(* CODESYS project DosingMachine (4).project

Project tree, tasks and I/O mapping:
  Device : CODESYS Control Win V3 x64, 3S - Smart Software Solutions GmbH, version 3.5.12.20
    application Application
      libraries: Standard, * (System); Util, * (System)
      task MainTask (cyclic, interval t#20ms, priority 1) calls DosingMain
      task VISU_TASK (cyclic, interval 100 ms, priority 31) calls VisuElems.Visu_Prg
      function block Timer [LD]
      function block DosingBlock [ST]
      program DosingMain [CFC]: Animatoin
      function block FSM [ST]
      visualisation Visualization
      image pool ImagePool
  text list GlobalTextList
  5ce3da45-db07-42e7-a21c-a00fff4ed8f6|E:\MyFiles\VideoShooting\CircuitBreakers\Slides\11.A to Z Project #2\PLC Porgramming\Motor 5.png
  5ce3da45-db07-42e7-a21c-a00fff4ed8f6|E:\MyFiles\VideoShooting\CircuitBreakers\Slides\11.A to Z Project #2\PLC Porgramming\helezon.png
  5ce3da45-db07-42e7-a21c-a00fff4ed8f6|E:\MyFiles\VideoShooting\CircuitBreakers\Slides\11.A to Z Project #2\helezon.png
  5ce3da45-db07-42e7-a21c-a00fff4ed8f6|E:\MyFiles\VideoShooting\CircuitBreakers\Slides\11.A to Z Project #2\PLC Porgramming\ELAVATOR 9 METRE - Kopya.PNG
  5ce3da45-db07-42e7-a21c-a00fff4ed8f6|E:\MyFiles\VideoShooting\CircuitBreakers\Slides\11.A to Z Project #2\Motor 5green.png
  5ce3da45-db07-42e7-a21c-a00fff4ed8f6|E:\MyFiles\VideoShooting\CircuitBreakers\Slides\11.A to Z Project #2\PLC Porgramming\Motor 5green.png
  5ce3da45-db07-42e7-a21c-a00fff4ed8f6|E:\MyFiles\VideoShooting\CircuitBreakers\Slides\11.A to Z Project #2\PLC Porgramming\Motor 5red.png
  5ce3da45-db07-42e7-a21c-a00fff4ed8f6|E:\MyFiles\VideoShooting\CircuitBreakers\Slides\11.A to Z Project #2\PLC Porgramming\ELAVATOR 9 METREFlip.png
  5ce3da45-db07-42e7-a21c-a00fff4ed8f6|E:\MyFiles\VideoShooting\CircuitBreakers\Slides\11.A to Z Project #2\PLC Porgramming\helezonFlip.png
  5ce3da45-db07-42e7-a21c-a00fff4ed8f6|E:\MyFiles\VideoShooting\CircuitBreakers\Slides\11.A to Z Project #2\PLC Porgramming\Silo.png
  5ce3da45-db07-42e7-a21c-a00fff4ed8f6|E:\MyFiles\VideoShooting\CircuitBreakers\Slides\11.A to Z Project #2\PLC Porgramming\Motor 5Flip.png
  5ce3da45-db07-42e7-a21c-a00fff4ed8f6|E:\MyFiles\VideoShooting\CircuitBreakers\Slides\11.A to Z Project #2\PLC Porgramming\Motor 5greenFlip.png
  5ce3da45-db07-42e7-a21c-a00fff4ed8f6|E:\MyFiles\VideoShooting\CircuitBreakers\Slides\11.A to Z Project #2\PLC Porgramming\Motor 5redflip.png
*)

// Device/Application/DosingMain
PROGRAM DosingMain
VAR
	Elev1Coil		:BOOL;
	Elev2Coil		:BOOL;
	Spiral1Coil		:BOOL;
	Spiral2Coil		:BOOL;
	MixerCoil		:BOOL;
	MixerGateCoil	:BOOL;
	
	Elev1OVLD		:BOOL;
	Elev2OVLD		:BOOL;
	SPiral1OVLD		:BOOL;
	Spiral2OVLD		:BOOL;
	MixerOVLD		:BOOL;
	EMGC			:BOOL;
	X: BOOL;
	StartDosing		:BOOL;
	StopDosing		:BOOL;
	FillSilo1		:BOOL;
	FillSilo2		:BOOL;
	
	Spiral1Freq		:INT;
	Spiral2Freq		:INT;
	MixerFreq		:INT;
	
	
	Silo1Weight		:INT;
	Silo2Weight		:INT;
	
	Silo1Required	:INT;
	Silo2Required	:INT;
	

	Silo1Dosing: DosingBlock;
	Silo2Dosing: DosingBlock;
	TheMaestro: FSM;
	Timing: Timer;
	LIN_TRAFO_0: lin_trafo;
	Silo1: LIN_TRAFO;
	Silo1Animation: WORD;
	Silo1AnimationScale: WORD;
	Silo2: LIN_TRAFO;
	Silo2Animation: WORD;
	Silo2AnimationScale: WORD;
END_VAR
VAR // added by the converter: edge detectors and wires of the graphical bodies
    _w1, _w2, _w3, _w16 : BOOL;
    _w4, _w5, _w6, _w7, _w8, _w9, _w10, _w11, _w12, _w13, _w14, _w15 : ANY;
END_VAR

Spiral2Coil := Silo2Dosing.MotorCoil;
MixerGateCoil := _w1;
_w3 := _w2 OR MixerOVLD;
Elev1Coil := FillSilo1;
Elev2Coil := FillSilo2;
Animatoin();
Silo1Dosing(
    StartDosing := _w4,
    StopDosing := StopDosing,
    Weight := Silo1Weight,
    RequiredProduct := Silo1Required); // DosingBlock
Spiral1Coil := Silo1Dosing.MotorCoil;
(* _w3 OR EMGC; result not used *)
Timing(MixerTimerActivate := _w5, GateTimerActivate := _w6, MixerPreSet := t#20s, GatePreSet := T#20s); // Timer
TheMaestro(
    Start := StartDosing,
    Stop := StopDosing,
    EMGC := _w7,
    Silo1DoseDone := _w8,
    Silo2DoseDone := _w9,
    Silo1NotEnough := _w10,
    Silo2NotEnough := _w11,
    FillBusy := _w12,
    MixerTimerDone := _w13,
    GateTimerDone := _w14); // FSM
Silo2Dosing(
    StartDosing := _w15,
    StopDosing := StopDosing,
    Weight := Silo2Weight,
    RequiredProduct := Silo2Required); // DosingBlock
_w12 := FillSilo1 OR FillSilo2;
MixerCoil := _w16;
_w2 := SPiral1OVLD OR Spiral2OVLD;

ACTION Animatoin:
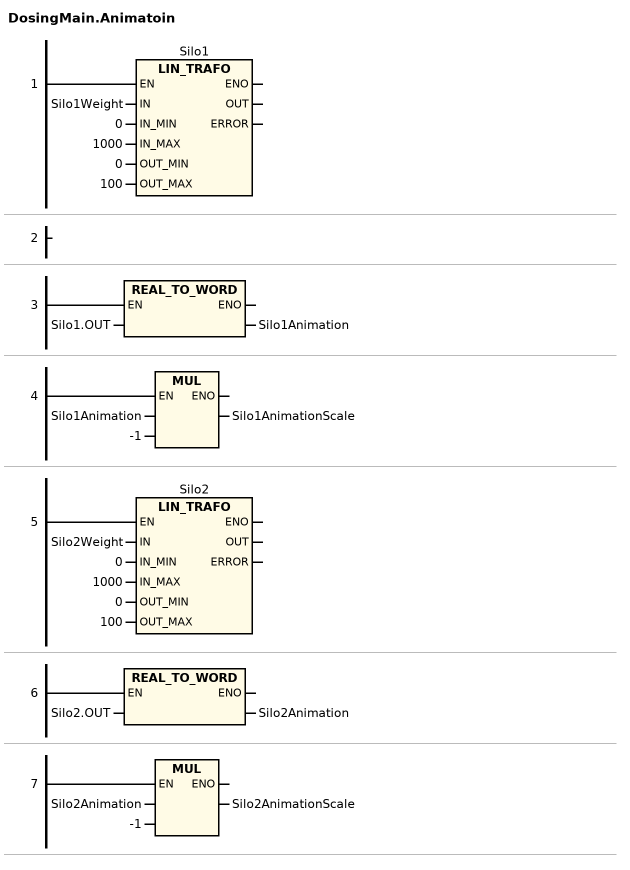
// NETWORK 1
Silo1(IN := Silo1Weight, IN_MIN := 0, IN_MAX := 1000, OUT_MIN := 0, OUT_MAX := 100); // LIN_TRAFO

// NETWORK 2

// NETWORK 3
Silo1Animation := REAL_TO_WORD(Silo1.OUT);

// NETWORK 4
Silo1AnimationScale := Silo1Animation * -1;

// NETWORK 5
Silo2(IN := Silo2Weight, IN_MIN := 0, IN_MAX := 1000, OUT_MIN := 0, OUT_MAX := 100); // LIN_TRAFO

// NETWORK 6
Silo2Animation := REAL_TO_WORD(Silo2.OUT);

// NETWORK 7
Silo2AnimationScale := Silo2Animation * -1;
END_ACTION

END_PROGRAM

// Device/Application/DosingBlock
FUNCTION_BLOCK DosingBlock
VAR_INPUT
	StartDosing : BOOL;
	StopDosing	: BOOL;
	Weight		:INT;
	RequiredProduct : INT;
	
END_VAR
VAR_OUTPUT
	MotorCoil        :BOOL;
	Extracted		 :INT;
	Busy			 :BOOL;
	Done			 :BOOL;
	NotEnough		 :BOOL;
END_VAR
VAR
	WeightSaved  : INT;
	StartTrig: R_TRIG;
END_VAR

StartTrig(CLK:=StartDosing , Q=> );

IF StartTrig.Q = 1 AND NotEnough=0 AND StopDosing=0 THEN
	WeightSaved := Weight ;
	MotorCoil:=1;
	Busy  :=1;
	Done :=0;
	
END_IF

IF Busy=1 THEN

Extracted :=	WeightSaved-Weight ;
IF Extracted>=RequiredProduct THEN
	MotorCoil :=0;
	Busy:=0;
	Done:=1;
END_IF
END_IF




IF RequiredProduct > Weight AND BUSY=0 THEN
	NotEnough:=1;
ELSE
	NotEnough:=0;
	
END_IF

IF StopDosing =1 THEN
	MotorCoil:=0;
	Busy:=0;
	Done:=1;
	
END_IF

END_FUNCTION_BLOCK

// Device/Application/Timer
FUNCTION_BLOCK Timer
VAR_INPUT
	MixerTimerActivate : BOOL;
	GateTimerActivate  :BOOL;
	MixerPreSet			:TIME;
	GatePreSet 			:TIME;
END_VAR
VAR_OUTPUT
	MixerTimerDone : BOOL;
	GateTimerDone   :BOOL;
END_VAR
VAR
	MixerTimer: TON;
	GateTimer: TON;
END_VAR

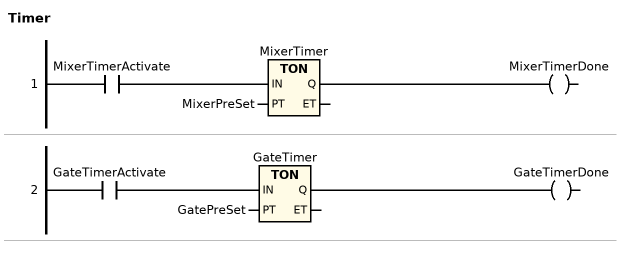
// NETWORK 1
MixerTimer(IN := MixerTimerActivate, PT := MixerPreSet); // TON
MixerTimerDone := MixerTimer.Q;

// NETWORK 2
GateTimer(IN := GateTimerActivate, PT := GatePreSet); // TON
GateTimerDone := GateTimer.Q;

END_FUNCTION_BLOCK

// Device/Application/FSM
FUNCTION_BLOCK FSM
VAR_INPUT
	Start 			:BOOL;
	Stop  			:BOOL;
	EMGC  			:BOOL;
	Silo1DoseDone 	:BOOL;
	Silo2DoseDone   :BOOL;
	Silo1NotEnough  :BOOL;
	Silo2NotEnough  :BOOL;
	FillBusy		:BOOL;
	MixerTimerDone  :BOOL;
	GateTimerDone	:BOOL;
	
END_VAR
VAR_OUTPUT
	Dose1BlockActivate  : BOOL;
	Dose2BlockActivate  :BOOL;
	MixerCoil		    :BOOL;
	GateCoil			:BOOL;
	MixerTimerActivate  :BOOL;
	GateTimerActivate   :BOOL;
	NotReady 			:BOOL;
	Stage				:INT;
END_VAR
VAR
	StartTrigger: R_TRIG;
	WeightSaved : INT;
	Silo1DoneTirg: R_TRIG;
	Silo2DoneTrig: R_TRIG;
END_VAR

StartTrigger(CLK:= Start , Q=> );
 
Silo1DoneTirg(CLK:= Silo1DoseDone  , Q=> );

 Silo2DoneTrig(CLK:= Silo2DoseDone , Q=> );
CASE Stage OF
	
0:
IF StartTrigger.Q = 1 AND NotReady=0 THEN
	Stage:=1;
END_IF

1:
Dose1BlockActivate:=1;
IF Silo1DoneTirg.Q =1 THEN
	Dose1BlockActivate:=0;
	Stage:=2;
END_IF

2:

Dose2BlockActivate:=1;
IF Silo2DoneTrig.Q =1 THEN
	Dose2BlockActivate:=0;
	Stage:=3;
END_IF


3:

MixerCoil:=1;
MixerTimerActivate:=1;

IF MixerTimerDone =1 THEN
MixerCoil:=0;
MixerTimerActivate:=0;	
Stage :=4;
END_IF

4:

GateCoil :=1 ;
GateTimerActivate := 1;
IF GateTimerDone =1 THEN
GateCoil :=0 ;	
GateTimerActivate := 0;
Stage:=0;

END_IF
END_CASE


IF EMGC OR Silo1NotEnough OR Silo2NotEnough OR FillBusy  OR STOP THEN
	NotReady :=1;
	MixerCoil:=0;
	GateCoil:=0;
	Dose1BlockActivate:=0;
	Dose2BlockActivate:=0;
	MixerTimerActivate:=0;
	GateTimerActivate :=0;
	Stage:=0;
	
ELSE
	NotReady:=0;
END_IF

END_FUNCTION_BLOCK

// Device/Application/Visualization
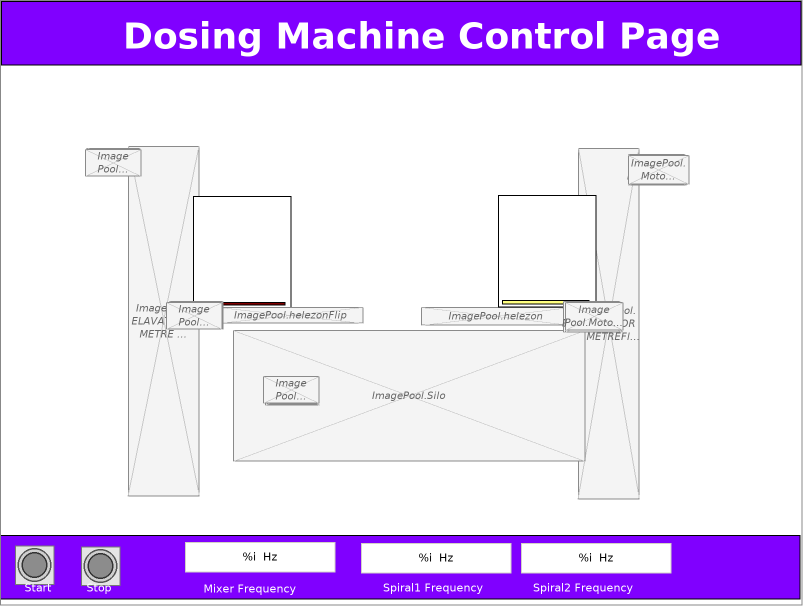
VISUALIZATION Visualization  // 803x606
    Rectangle (1,1 800x64)
    Label (105,9 634x54), "Dosing Machine Control Page"
    Rectangle (0,535 800x64)
    PushSwitch (15,540 39x50), variable: DosingMain.StartDosing, behaviour: TAP, style: Switch-PushSwitch-Gray
    PushSwitch (81,541 39x50), variable: DosingMain.StopDosing, behaviour: TAP, style: Switch-PushSwitch-Gray
    Label (-37,573 150x30), "Start"
    Label (24,573 150x30), "Stop"
    Textfield (521,543 150x30), "%i Hz", text variable: DosingMain.Spiral2Freq
    Textfield (361,543 150x30), "%i Hz", text variable: DosingMain.Spiral1Freq
    Textfield (185,542 150x30), "%i Hz", text variable: DosingMain.MixerFreq
    Label (175,574 150x30), "Mixer Frequency"
    Label (358,573 150x30), "Spiral1 Frequency"
    Label (508,573 150x30), "Spiral2 Frequency"
    Image (128,146 71x350), image: ImagePool.ELAVATOR 9 METRE - Kopya
    Image (578,148 61x351), image: ImagePool.ELAVATOR 9 METREFlip0
    Image (421,307 150x18), image: ImagePool.helezon
    Rectangle (193,196 98x112)
    Image (218,307 145x16), image: ImagePool.helezonFlip
    Image (233,330 352x131), image: ImagePool.Silo
    Rectangle (498,195 98x112)
    RoundedRectangle (198,302 87x3)
        p2773130477: DosingMain.Silo2AnimationScale
    RoundedRectangle (502,300 87x4)
        p2773130477: DosingMain.Silo1AnimationScale
    Image (86,148 54x28), image: ImagePool.Motor 5
    Image (88,148 52x26), invisible if: DosingMain.Elev1Coil=0, image: ImagePool.Motor 5green
    Image (85,149 56x27), invisible if: DosingMain.Elev1OVLD=0, image: ImagePool.Motor 5red
    Image (169,301 54x28), image: ImagePool.Motor 5
    Image (169,302 52x26), invisible if: DosingMain.Spiral2Coil=0, image: ImagePool.Motor 5green
    Image (166,302 56x27), invisible if: DosingMain.Spiral2OVLD=0, image: ImagePool.Motor 5red
    Image (265,377 54x28), image: ImagePool.Motor 5
    Image (267,378 52x26), invisible if: DosingMain.MixerCoil=0, image: ImagePool.Motor 5green
    Image (263,376 56x27), invisible if: DosingMain.MixerOVLD=0, image: ImagePool.Motor 5red
    Image (628,154 57x31), image: ImagePool.Motor 5Flip
    Image (629,155 57x30), invisible if: DosingMain.Elev2Coil=0, image: ImagePool.Motor 5greenFlip
    Image (628,155 61x29), invisible if: DosingMain.Elev2OVLD=0, image: ImagePool.Motor 5redflip
    Image (563,301 57x31), image: ImagePool.Motor 5Flip
    Image (565,302 57x30), invisible if: DosingMain.Spiral1Coil=0, image: ImagePool.Motor 5greenFlip
    Image (565,302 58x28), invisible if: DosingMain.SPiral1OVLD=0, image: ImagePool.Motor 5redflip
END_VISUALIZATION
